PROGRAM VisuComments
VAR
END_VAR

(*
//Visu consist of 2 frames:
	- Object browser	- used for browsing the object tree. It is possible to access every
						object through it. Side buttons are used to move between syblings.
						Buttons above and below current object name help to move between generations.
						Enter the name of the object on the middle and clikc 'Search' to find any object.
						
						- 'Change param' opens dialog that can be used to modify internal value of any object
						implementing I_Param interface. Use 'Copy Param from browser' each time the value or active object changed.
	
	- Logs				- contain all events, such as add or remove child, attach sub/pub, update sub, etc.


*)

END_PROGRAM

(* stored: Version 1.1.0.1, ProductVersion 3.1.4024.12
   POU VisuComments: Id {0a4cbecb-741e-436a-bb74-3baa223f060d}, SpecialFunc None *)
